TYPE ST_SectorConfig :
STRUCT
	TrackObjectId			: OTCID;
	PartObjectId	    : OTCID;
	PartObjectIdEnt	    : OTCID;
	PartObjectIdExit    : OTCID;	
	PartSectorStartPosn				: LREAL;
	PartSectorEndPosn				: LREAL;
	TrackSectorStartPosn				: LREAL;
	TrackSectorEndPosn				: LREAL;
	SectorSpansBoundary		: BOOL;
END_STRUCT
END_TYPE

(* stored: Version 1.1.0.1, ProductVersion 3.1.4026.8
   DUT ST_SectorConfig: Id {77932430-4813-013f-16b4-5b3df9147ac2} *)
